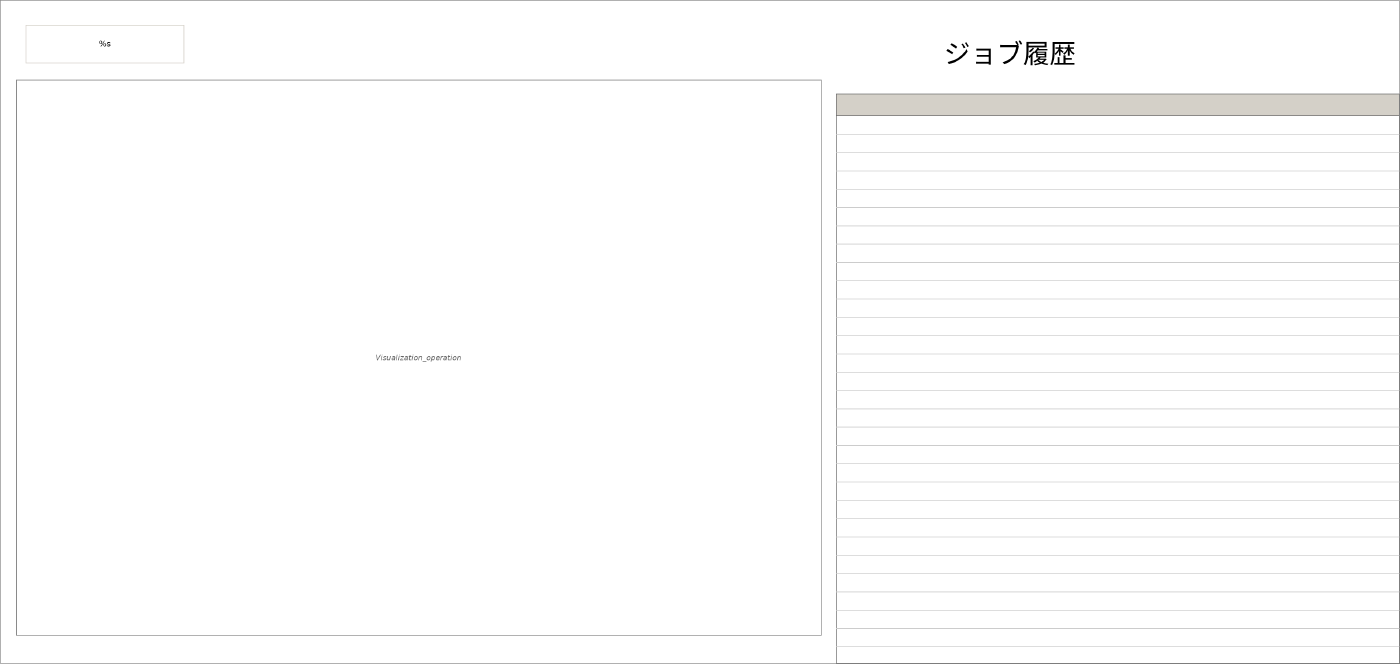
VISUALIZATION Visualization  // 1911x907
    TabControl (22,109 1099x759)
        shows Visualization_operation()
        shows Visualization_recipe()
        [0]: TabTitle=メイン
        [1]: TabTitle=マニュアル動作
    Table (1141,128 770x779), data array: MAIN.ads_reporter.log_view
        p3854506369: MAIN.ads_reporter.log_view[0,INDEX]
        p1892666644: MAIN.ads_reporter.log_view[1,INDEX]
        p2232123230: 時刻
        p511219082: タスク名
        p2685023577: MAIN.ads_reporter.log_view[INDEX]
        p338671338: MAIN.ads_reporter.log_view[3,INDEX]
        p1755163831: ジョブID
        p2170511999: MAIN.ads_reporter.log_view[2,INDEX]
        p4092479075: イベント
    Label (1164,50 429x47), "ジョブ履歴"
    Textfield (35,34 216x52), "%s", text list: 'MachineMode', text index: MAIN.machine_mode
END_VISUALIZATION

(* stored: Version 1.1.0.1, ProductVersion 3.1.4024.12
   Visu Visualization: Id {270ba47c-d781-43fd-82fc-92e2d7d2e42e} *)
